Fanuc KAREL source: kt00066.KL

-- PROVISIONAL review KL for V770-1; original PC SHA256 c067c702051e004f664249f2fef945c988d272684d26c895f2607e77ee22fb04
-- Incomplete behavior may be omitted. Consult companion uncertainty JSON. Do not deploy.
PROGRAM KT00066
%NOLOCKGROUP
VAR
  I1 : INTEGER
  I2 : INTEGER
  OUT : REAL
BEGIN
  -- UNRESOLVED_PC offsets 5-16; opcodes 2E,23
  -- UNRESOLVED_PC offsets 21-32; opcodes 2E,23
  -- UNRESOLVED_PC offsets 37-48; opcodes 2E,23
  -- UNRESOLVED_PC offsets 53-64; opcodes 2E,23
  -- UNRESOLVED_PC offsets 69-89; opcodes 21,21,54,64,23
  -- UNRESOLVED_PC offsets 94-98; opcodes 7F
END KT00066
